// TIA Portal V19 export
TYPE "type_u3RequestData"
// stored: Access Published, Namespace Unit3
   STRUCT
      u3ToxyzU1Transfered : Bool;   // 允许运动
      u3ToxyzU2Transfered : Bool;   // 允许运动
   END_STRUCT;
END_TYPE
